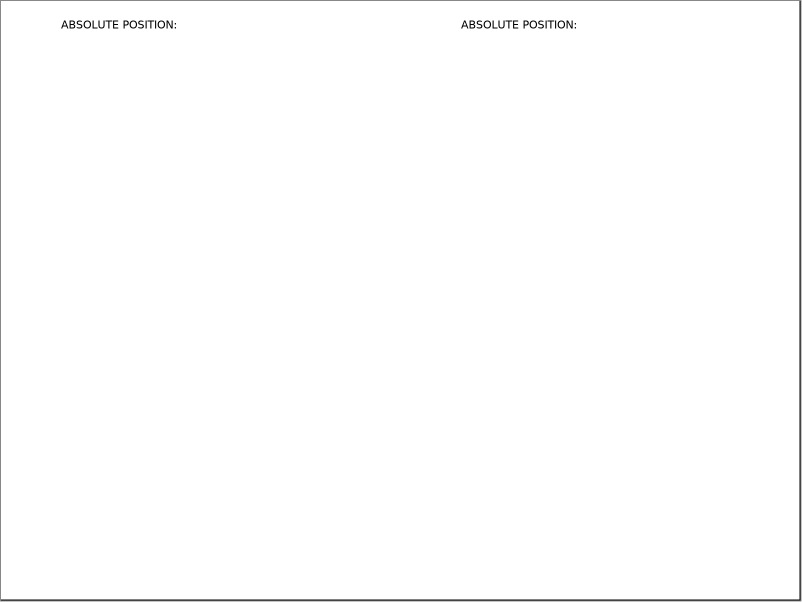
VISUALIZATION F17_Set_Position  // 802x602
    Rectangle (0,0 800x600)
    Label (10,10 170x30), "ABSOLUTE POSITION:"
    Label (410,10 170x30), "ABSOLUTE POSITION:"
END_VISUALIZATION

(* stored: Version 1.1.0.1, ProductVersion 3.1.4022.7
   Visu F17_Set_Position: Id {03599216-c009-41f1-87c8-6ac98b505f30} *)
